{attribute 'qualified_only'}
{attribute 'strict'}
TYPE E_VELOCITY_STATE_MACHINE :
(
	POWER_OFF := 0,
	POWER_ON := 1,
	VELOCITY := 2 
);
END_TYPE

(* stored: Version 1.1.0.1, ProductVersion 3.1.4022.3
   DUT E_VELOCITY_STATE_MACHINE: Id {6e646859-0427-4e9a-9e5e-ca8eb1bd3d9b} *)
